TYPE ST_Inputs :
STRUCT
	// CAN
	Inputs 				AT %I*	: CANRXQUEUESTRUCT_N_1;
	
	// IO
	nEL3702Ch1_In 		AT %I*	: INT;
	nEL3702Ch2_In 		AT %I*	: INT;
	nEL3702Ch3_In 		AT %I*	: INT;
	
	// Encoder
	nEL5101_Counter 	AT %I*	: UINT;
	bEL5101_CounterSet	AT %I*	: BIT;
	nEL5101_LatchValue	AT %I*	: UINT;
	nEL5101_Frequency	AT %I*	: UDINT;
	bEL5101_LatchValid	AT %I*	: BIT;
	
	// From controller
	fAlpha_U, fBeta_U	AT %I*	: LREAL;
	iQ, iD				AT %I*	: LREAL;
END_STRUCT
END_TYPE

(* stored: Version 1.1.0.1, ProductVersion 3.1.4024.11
   DUT ST_Inputs: Id {39d9a656-d2dc-42a1-b92e-092053ce1266} *)
